// Mitsubishi GX Works2 project: BookEX6_12 Counter   PLC: Q13UDV

// global labels: Global
VAR_GLOBAL
  bVar0 AT M5000 : BOOL;
  abArray0 AT M5010 : ARRAY [0..49] OF BOOL;
  sStr0 AT D5000 : STRING[199];
  sStr1 AT D5100 : STRING[199];
  sStr2 AT D5200 : STRING[199];
  sStr3 AT D5300 : STRING[199];
  sStr4 AT D5400 : STRING[199];
  sStr5 AT D5500 : STRING[199];
  sStr6 AT D5600 : STRING[199];
  sStr7 AT D5700 : STRING[199];
  sStr8 AT D5800 : STRING[199];
  sStr9 AT D5900 : STRING[199];
  iVar0 AT D4500 : INT;
  iVar1 AT D4501 : INT;
  iVar2 AT D4502 : INT;
  iVar3 AT D4503 : INT;
  iVar4 AT D4504 : INT;
  iVar5 AT D4505 : INT;
  iVar6 AT D4506 : INT;
  iVar7 AT D4507 : INT;
  iVar8 AT D4508 : INT;
  iVar9 AT D4509 : INT;
  dVar0 AT D4510 : DINT;
  dVar1 AT D4512 : DINT;
  dVar2 AT D4514 : DINT;
  dVar3 AT D4516 : DINT;
  dVar4 AT D4518 : DINT;
  dVar5 AT D4520 : DINT;
  dVar6 AT D4522 : DINT;
  dVar7 AT D4524 : DINT;
  dVar8 AT D4526 : DINT;
  dVar9 AT D4528 : DINT;
  wVar0 AT D4530 : WORD;
  wVar1 AT D4531 : WORD;
  wVar2 AT D4532 : WORD;
  wVar3 AT D4533 : WORD;
  wVar4 AT D4534 : WORD;
  wVar5 AT D4535 : WORD;
  wVar6 AT D4536 : WORD;
  wVar7 AT D4537 : WORD;
  wVar8 AT D4538 : WORD;
  wVar9 AT D4539 : WORD;
  dwVar0 AT D4540 : DWORD;
  dwVar1 AT D4542 : DWORD;
  dwVar2 AT D4544 : DWORD;
  dwVar3 AT D4546 : DWORD;
  dwVar4 AT D4548 : DWORD;
  dwVar5 AT D4550 : DWORD;
  dwVar6 AT D4552 : DWORD;
  dwVar7 AT D4554 : DWORD;
  dwVar8 AT D4556 : DWORD;
  dwVar9 AT D4558 : DWORD;
  fsVar0 AT D4560 : REAL;
  fsVar1 AT D4562 : REAL;
  fsVar2 AT D4564 : REAL;
  fsVar3 AT D4566 : REAL;
  fsVar4 AT D4568 : REAL;
  fsVar5 AT D4570 : REAL;
  fsVar6 AT D4572 : REAL;
  fsVar7 AT D4574 : REAL;
  fsVar8 AT D4576 : REAL;
  fsVar9 AT D4578 : REAL;
  fdVar0 AT D4580 : LREAL;
  tTime0 AT D4620 : TIME;
  tTime1 AT D4622 : TIME;
  tTime2 AT D4624 : TIME;
  tTime3 AT D4626 : TIME;
  tTime4 AT D4628 : TIME;
  tTime5 AT D4630 : TIME;
  tTime6 AT D4632 : TIME;
  tTime7 AT D4634 : TIME;
  tTime8 AT D4636 : TIME;
  tTime9 AT D4638 : TIME;
  tTime10 AT D4640 : TIME;
  bVar1 AT M5001 : BOOL;
  bVar2 AT M5002 : BOOL;
  bVar3 AT M5003 : BOOL;
  bVar4 AT M5004 : BOOL;
  bVar5 AT M5005 : BOOL;
  bVar6 AT M5006 : BOOL;
  bVar7 AT M5007 : BOOL;
  bVar8 AT M5008 : BOOL;
  bVar9 AT M5009 : BOOL;
  abArray1 AT M5060 : ARRAY [0..49] OF BOOL;
  abArray2 AT M5110 : ARRAY [0..49] OF BOOL;
  abArray3 AT M5160 : ARRAY [0..49] OF BOOL;
  abArray4 AT M5210 : ARRAY [0..49] OF BOOL;
  abArray5 AT M5260 : ARRAY [0..49] OF BOOL;
  abArray6 AT M5310 : ARRAY [0..49] OF BOOL;
  abArray7 AT M5360 : ARRAY [0..49] OF BOOL;
  abArray8 AT M5410 : ARRAY [0..49] OF BOOL;
  abArray9 AT M5460 : ARRAY [0..49] OF BOOL;
  fdVar1 AT D4584 : LREAL;
  fdVar2 AT D4588 : LREAL;
  fdVar3 AT D4592 : LREAL;
  fdVar4 AT D4596 : LREAL;
  fdVar5 AT D4600 : LREAL;
  fdVar6 AT D4604 : LREAL;
  fdVar7 AT D4608 : LREAL;
  fdVar8 AT D4612 : LREAL;
  fdVar9 AT D4616 : LREAL;
  aSendData1 AT D100 : ARRAY [0..9] OF INT;
  aiTxData AT D4000 : ARRAY [0..99] OF INT;
  aiRxData AT D4100 : ARRAY [0..99] OF INT;
  iOpenOK AT D3900 : INT;
  iOpenERR AT D3901 : INT;
  iSendOK AT D3902 : INT;
  iSendERR AT D3903 : INT;
  iCloseOK AT D3906 : INT;
  iCloseERR AT D3907 : INT;
  iRecvOK AT D3904 : INT;
  iRecvERR AT D3905 : INT;
  aiTxData2 AT D4200 : ARRAY [0..99] OF INT;
  aiRxData2 AT D4300 : ARRAY [0..99] OF INT;
  iOpenOK2 AT D3908 : INT;
  iOpenERR2 AT D3909 : INT;
  iSendOK2 AT D3910 : INT;
  iSendERR2 AT D3911 : INT;
  iRecvOK2 AT D3912 : INT;
  iRecvERR2 AT D3913 : INT;
  iCloseOK2 AT D3914 : INT;
  iCloseERR2 AT D3915 : INT;
  iEOpenComp AT D3916 : INT;
  iEOpenReq AT D3917 : INT;
  iERecvFlag AT D3918 : INT;
  iOpenCode AT D3919 : INT;
  iSendCode AT D3920 : INT;
  iRecvCode AT D3921 : INT;
  iCloseCode AT D3922 : INT;
  iOpenCode2 AT D3923 : INT;
  iSendCode2 AT D3924 : INT;
  iRecvCode2 AT D3925 : INT;
  iCloseCode2 AT D3926 : INT;
  aRecvData1 AT D110 : ARRAY [0..9] OF INT;
  aSendData2 AT D120 : ARRAY [0..9] OF INT;
  aRecvData2 AT D130 : ARRAY [0..9] OF INT;
  CC1 : BOOL;
END_VAR
// user libraries (not included): HMI

FUNCTION_BLOCK newCTD
VAR_INPUT
  b_CD : BOOL;
  b_LOAD : BOOL;
END_VAR
VAR_OUTPUT
  b_Q : BOOL;
  i_CV : INT;
END_VAR
VAR_INPUT
  i_PV : INT;
END_VAR
;
IF b_LOAD THEN
	i_CV := i_PV;
ELSIF LDP(TRUE, b_CD) AND (i_CV > 0) THEN
	i_CV := i_CV - 1;
END_IF;
b_Q := i_CV <=  0;
END_FUNCTION_BLOCK

FUNCTION_BLOCK newCTU
VAR_INPUT
  b_CU : BOOL;
  b_RST : BOOL;
END_VAR
VAR_OUTPUT
  b_Q : BOOL;
  i_CV : INT;
END_VAR
VAR_INPUT
  i_PV : INT;
END_VAR
;
IF b_RST THEN
	i_CV := 0;
ELSIF LDP(TRUE, b_CU) AND (i_CV < i_PV) THEN
	i_CV := i_CV + 1;
END_IF;
b_Q := i_CV >= i_PV;
END_FUNCTION_BLOCK

FUNCTION_BLOCK newCTUD
VAR_INPUT
  b_CU : BOOL;
  b_RST : BOOL;
END_VAR
VAR_OUTPUT
  b_QU : BOOL;
  i_CV : INT;
END_VAR
VAR_INPUT
  i_PV : INT;
  b_CD : BOOL;
  b_LOAD : BOOL;
END_VAR
VAR_OUTPUT
  b_QD : BOOL;
END_VAR
;
IF b_RST THEN
	i_CV := 0;
ELSIF  b_LOAD THEN i_CV := i_PV;
ELSE
	IF LDP(TRUE, b_CU) AND (i_CV < i_PV) THEN
		i_CV := i_CV + 1;
	ELSIF LDP(TRUE, b_CD) AND (i_CV > 0) THEN
		i_CV := i_CV - 1;
	END_IF;
END_IF;
b_QU := i_CV >= i_PV;
b_QD := i_CV <= 0;
END_FUNCTION_BLOCK

PROGRAM ExCOUNT
VAR
  CTU_E_1 : CTU_E;
  COUNTER_FB_M_1 : COUNTER_FB_M;
  HMI15_1 : HMI15;
END_VAR
(* structured ladder/FBD written out as ST: instructions are called as NAME(EN, inputs, outputs); _pN, _eN, _tN stand for wires *)
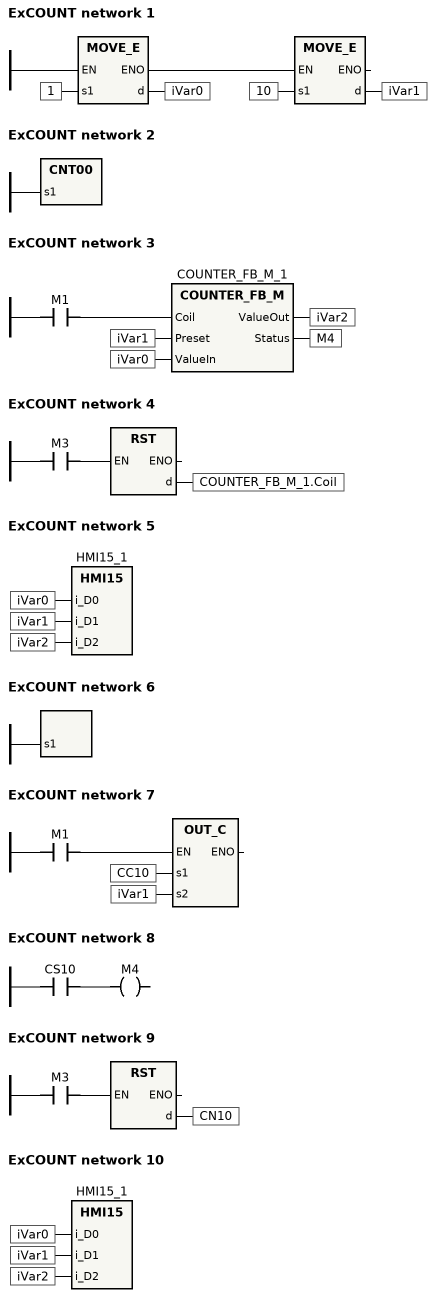
(* network 1 *)
_e1 := MOVE_E(TRUE, 1, iVar0);
MOVE_E(_e1, 10, iVar1);
(* network 2 *)
(* element kind 9 CNT00 <- TRUE *)
(* network 3 *)
COUNTER_FB_M_1(Coil := M1, Preset := iVar1, ValueIn := iVar0, ValueOut => iVar2, Status => M4);
(* network 4 *)
RST(M3, COUNTER_FB_M_1.Coil);
(* network 5 *)
HMI15_1(i_D0 := iVar0, i_D1 := iVar1, i_D2 := iVar2);
(* network 6 *)
(* element kind 10  <- TRUE *)
(* network 7 CNT00: *)
OUT_C(M1, CC10, iVar1);
(* network 8 *)
M4 := CS10;
(* network 9 *)
RST(M3, CN10);
(* network 10 *)
HMI15_1(i_D0 := iVar0, i_D1 := iVar1, i_D2 := iVar2);
END_PROGRAM

PROGRAM ExCTD
VAR
  CTD_E_1 : CTD_E;
  HMI15_1 : HMI15;
END_VAR
(* structured ladder/FBD written out as ST: instructions are called as NAME(EN, inputs, outputs); _pN, _eN, _tN stand for wires *)
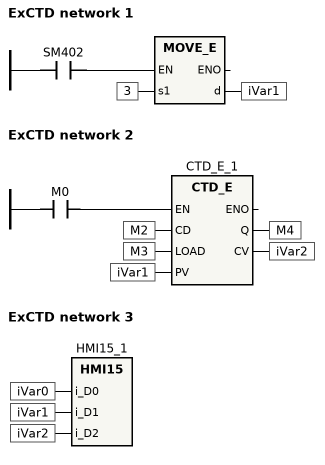
(* network 1 *)
MOVE_E(SM402, 3, iVar1);
(* network 2 *)
CTD_E_1(EN := M0, CD := M2, LOAD := M3, PV := iVar1, Q => M4, CV => iVar2);
(* network 3 *)
HMI15_1(i_D0 := iVar0, i_D1 := iVar1, i_D2 := iVar2);
END_PROGRAM

PROGRAM ExCTU
VAR
  CTU_E_1 : CTU_E;
  HMI15_1 : HMI15;
END_VAR
(* structured ladder/FBD written out as ST: instructions are called as NAME(EN, inputs, outputs); _pN, _eN, _tN stand for wires *)
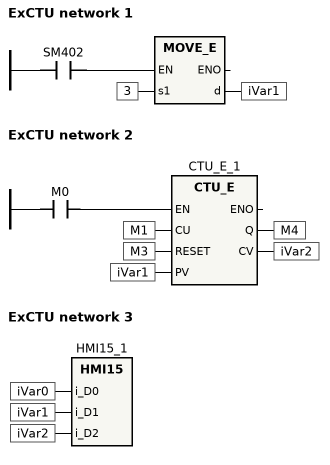
(* network 1 *)
MOVE_E(SM402, 3, iVar1);
(* network 2 *)
CTU_E_1(EN := M0, CU := M1, RESET := M3, PV := iVar1, Q => M4, CV => iVar2);
(* network 3 *)
HMI15_1(i_D0 := iVar0, i_D1 := iVar1, i_D2 := iVar2);
END_PROGRAM

PROGRAM ExCTUD
VAR
  CTUD_E_1 : CTUD_E;
  HMI15_1 : HMI15;
END_VAR
(* structured ladder/FBD written out as ST: instructions are called as NAME(EN, inputs, outputs); _pN, _eN, _tN stand for wires *)
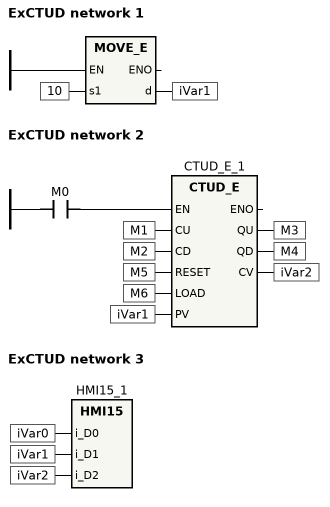
(* network 1 *)
MOVE_E(TRUE, 10, iVar1);
(* network 2 *)
CTUD_E_1(EN := M0, CU := M1, CD := M2, RESET := M5, LOAD := M6, PV := iVar1, QU => M3, QD => M4, CV => iVar2);
(* network 3 *)
HMI15_1(i_D0 := iVar0, i_D1 := iVar1, i_D2 := iVar2);
END_PROGRAM

PROGRAM ExNewCTD
VAR
  newCTD_1 : newCTD;
  HMI15_1 : HMI15;
END_VAR
(* structured ladder/FBD written out as ST: instructions are called as NAME(EN, inputs, outputs); _pN, _eN, _tN stand for wires *)
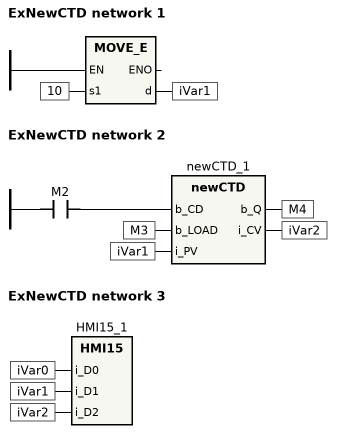
(* network 1 *)
MOVE_E(TRUE, 10, iVar1);
(* network 2 *)
newCTD_1(b_CD := M2, b_LOAD := M3, i_PV := iVar1, b_Q => M4, i_CV => iVar2);
(* network 3 *)
HMI15_1(i_D0 := iVar0, i_D1 := iVar1, i_D2 := iVar2);
END_PROGRAM

PROGRAM ExNewCTU
VAR
  newCTU_1 : newCTU;
  HMI15_1 : HMI15;
END_VAR
(* structured ladder/FBD written out as ST: instructions are called as NAME(EN, inputs, outputs); _pN, _eN, _tN stand for wires *)
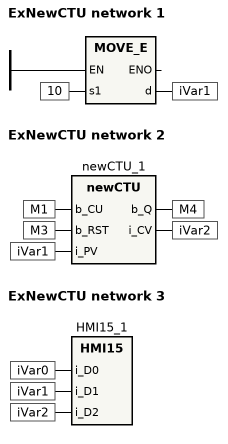
(* network 1 *)
MOVE_E(TRUE, 10, iVar1);
(* network 2 *)
newCTU_1(b_CU := M1, b_RST := M3, i_PV := iVar1, b_Q => M4, i_CV => iVar2);
(* network 3 *)
HMI15_1(i_D0 := iVar0, i_D1 := iVar1, i_D2 := iVar2);
END_PROGRAM

PROGRAM ExNewCTUD
VAR
  newCTUD_1 : newCTUD;
  HMI15_1 : HMI15;
END_VAR
(* structured ladder/FBD written out as ST: instructions are called as NAME(EN, inputs, outputs); _pN, _eN, _tN stand for wires *)
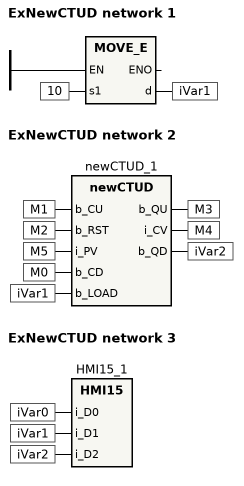
(* network 1 *)
MOVE_E(TRUE, 10, iVar1);
(* network 2 *)
newCTUD_1(b_CU := M1, b_RST := M2, i_PV := M5, b_CD := M0, b_LOAD := iVar1, b_QU => M3, i_CV => M4, b_QD => iVar2);
(* network 3 *)
HMI15_1(i_D0 := iVar0, i_D1 := iVar1, i_D2 := iVar2);
END_PROGRAM

PROGRAM ExCTU_ST
VAR
  fbCounter : CTU;
  bInput : BOOL;
  bReset : BOOL;
  bDone : BOOL;
  iCurrCounter : INT;
END_VAR
;


fbCounter(CU := bInput, RESET := bReset, PV := 5); 	(* 입력 조건만 넣고 카운터 실행*)

IF fbCounter.Q THEN														(* 필요한 곳에서출력값 호출*)
    bDone := TRUE;														(* 5회 카운트시 실행할 로직*)
END_IF;

iCurrCounter := fbCounter.CV;										(* 현재 값*)
END_PROGRAM

PROGRAM ExCTD_ST
VAR
  fbCounter : CTD;
  bInput : BOOL;
  bLoad : BOOL;
  bDone : BOOL;
  iCurrCounter : INT;
END_VAR


fbCounter(CD := bInput AND NOT fbCounter.Q , LOAD := bLoad, PV := 5); 	

IF fbCounter.Q THEN														(* 필요한 곳에서출력값 호출*)
    bDone := TRUE;														(* 5회 카운트시 실행할 로직*)
END_IF;

iCurrCounter := fbCounter.CV;										(* 현재 값*);
END_PROGRAM

PROGRAM ExCTUD_ST
VAR
  fbCounter : CTUD;
  bEnter : BOOL;
  bLoad : BOOL;
  bFull : BOOL;
  iCurrCounter : INT;
  bReset : BOOL;
  bExit : BOOL;
  bEmpty : BOOL;
END_VAR
;


fbCounter(CU := bEnter AND NOT fbCounter.QU , CD := bExit AND NOT fbCounter.QD , 
					RESET := bReset, LOAD := bReset, PV := 5); 	

bFull := fbCounter.QU;
bEmpty := fbCounter.QD;

iCurrCounter := fbCounter.CV;					(* 현재 주차차량*);
END_PROGRAM

PROGRAM ExOut_C
VAR
  HMI05_1 : HMI05;
END_VAR
(* structured ladder/FBD written out as ST: instructions are called as NAME(EN, inputs, outputs); _pN, _eN, _tN stand for wires *)
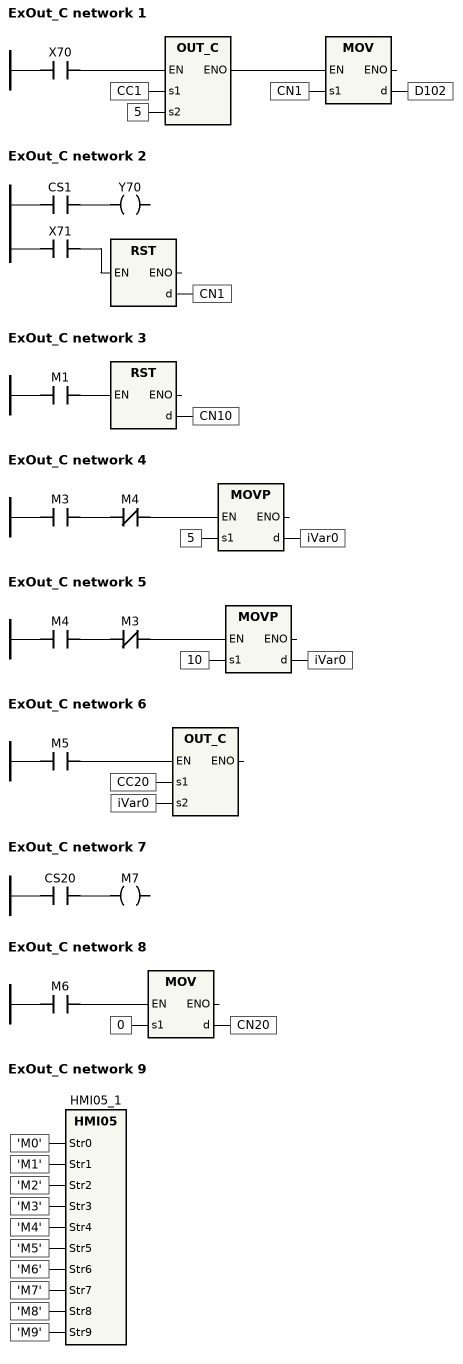
(* network 1 *)
_e1 := OUT_C(X70, CC1, 5);
MOV(_e1, CN1, D102);
(* network 2 *)
Y70 := CS1;
RST(X71, CN1);
(* network 3 *)
RST(M1, CN10);
(* network 4 *)
MOVP(M3 AND NOT M4, 5, iVar0);
(* network 5 *)
MOVP(M4 AND NOT M3, 10, iVar0);
(* network 6 *)
OUT_C(M5, CC20, iVar0);
(* network 7 *)
M7 := CS20;
(* network 8 *)
MOV(M6, 0, CN20);
(* network 9 *)
HMI05_1(Str0 := 'M0', Str1 := 'M1', Str2 := 'M2', Str3 := 'M3', Str4 := 'M4', Str5 := 'M5', Str6 := 'M6', Str7 := 'M7', Str8 := 'M8', Str9 := 'M9');
END_PROGRAM
